{attribute 'linkalways'} 
{attribute 'no_explicit_call' := 'This FB is a CLASS and must be accessed using methods or properties'}
{attribute 'enable_dynamic_creation'}
FUNCTION_BLOCK Node_F_VN_DrawPoints EXTENDS VisionNode
VAR
    ipPoints : _ITcVnContainer;
    ipDestImage : _ITcVnImage;
    eShape : _ETcVnDrawShape(ETcVnDrawShape.TCVN_DS_CIRCLE);
    aColor : _TcVnVector4_LREAL;
    hrPrev : _HRESULT(S_OK);
	hresult : _HRESULT(S_OK);
END_VAR

METHOD PUBLIC  Clone : I_Node
VAR
	pNode : POINTER TO Node_F_VN_DrawPoints;
END_VAR
pNode := __NEW(Node_F_VN_DrawPoints);
Clone := pNode^;
END_METHOD

METHOD FB_init : BOOL
VAR_INPUT
	bInitRetains : BOOL; // if TRUE, the retain variables are initialized (warm start / cold start)
	bInCopyCode : BOOL;  // if TRUE, the instance afterwards gets moved into the copy code (online change)
END_VAR
AddInput('ipPoints', ipPoints);
AddInput('ipDestImage', ipDestImage);
AddParameter('eShape', eShape);
AddInput('aColor', aColor);
AddInput('hrPrev', hrPrev);
AddOutput('ipDestImage', ipDestImage);
AddOutput('hresult',hresult);
END_METHOD

METHOD PROTECTED OnExecute
hresult.Value := F_VN_DrawPoints(
    ipPoints := ipPoints.Value,
	ipDestImage := ipDestImage.Value,
    eShape := eShape.Value,
    aColor := aColor.Value,
	hrPrev:= hrPrev.Value);
END_METHOD

METHOD PUBLIC PreExecutionCheck
VAR_INPUT
	Check : I_PreExecutionChecks;
END_VAR
Check.IsTrue(ipPoints.IsValid, 'ipPoints must be a valid container');
Check.IsTrue((ipPoints.IsType(TC_GLOBAL_CONST_LIST.ContainerType_Vector_TcVnPoint2_DINT) OR
              ipPoints.IsType(TC_GLOBAL_CONST_LIST.ContainerType_Vector_TcVnPoint2_REAL)),
              'ipPoints contains incorrect type');
              
Check.IsTrue(ipDestImage.IsValid, 'ipDestImage must contain an image');
END_METHOD

END_FUNCTION_BLOCK

(* stored: Version 1.1.0.1, ProductVersion 3.1.4026.13
   POU Node_F_VN_DrawPoints: Id {21f961e9-ab7f-041f-0325-035b95434fed}, SpecialFunc None
   Folder Constructor: Id {fb84f928-1693-0621-3c4b-5cc3b866e1b5}
   Method Clone: Id {7589a694-a049-0b33-2e4c-2d8defbb3e7a}
   Method FB_init: Id {ef6d4d23-ac9c-0ba4-3a6f-7984cd801e40}
   Method OnExecute: Id {d405b788-6b1a-0e0c-1710-dfbb159c71c4}
   Method PreExecutionCheck: Id {2383b19f-fb8a-0fda-226a-f63f3a8f62d2} *)
